// TIA Portal V20 export
// export: Created 2025-12-01T14:56:16.2448627Z, ExportSetting None, DisplayName Totally Integrated Automation Portal, DisplayVersion V20 Update 3, DisplayName TIA Portal Openness, DisplayVersion V20 Update 3, DisplayName TIA Portal Version Control Interface, DisplayVersion V20 Update 3, DisplayName STEP 7 Professional, DisplayVersion V20 Update 3, DisplayName STEP 7 Safety, DisplayVersion V20 Update 2, DisplayName WinCC Basic/Comfort/Advanced, DisplayVersion V20 Update 3, DisplayName WinCC Professional, DisplayVersion V20 Update 3, DisplayName WinCC Unified, DisplayVersion V20 Update 3
TYPE "ROUT_Estadisticas_Scanners"
   STRUCT
      Lect_Good : UInt;
      Lect_NoGood : UInt;
      Lect_NoFound : UInt;
      Lect_NoGood_consecutivas : UInt;
      Porcentaje_error_lecturas : UInt;
   END_STRUCT;
END_TYPE
